(* Logix 5000 project; controller reports 1756-L63 rev 20.11; software revision 20.04; part 51 of 52 *)

        [192].log_data[2].total := 459.251, [192].log_data[2].time := 3600.0, [192].log_data[2].minminute := 7, [192].log_data[2].valid := 1, [192].log_data[3].time := 3600.0, [192].log_data[3].valid := 1, [192].log_data[4].time := 3600.0, [192].log_data[4].valid := 1, [192].log_data[5].max := 1.0, [192].log_data[5].total := 245.0, [192].log_data[5].time := 3600.0, [192].log_data[5].maxminute := 1, [192].log_data[5].valid := 1, [192].log_data[6].time := 3600.0, [192].log_data[6].valid := 1, [192].log_data[7].time := 3600.0, [192].log_data[7].valid := 1, [192].log_data[8].max := 1.0, [192].log_data[8].total := 3412.249, [192].log_data[8].time := 3600.0, [192].log_data[8].maxminute := 3, [192].log_data[8].valid := 1, [192].log_data[9].max := 1.0, [192].log_data[9].total := 3408.749, [192].log_data[9].time := 3600.0, [192].log_data[9].maxminute := 3, [192].log_data[9].valid := 1, [192].log_data[10].min := 1.0, [192].log_data[10].max := 1.0, [192].log_data[10].total := 3600.0, [192].log_data[10].time := 3600.0, [192].log_data[10].valid := 1, [192].log_data[11].time := 3600.0, [192].log_data[11].valid := 1, [192].log_data[12].min := 1.0, [192].log_data[12].max := 1.0, [192].log_data[12].total := 3600.0, [192].log_data[12].time := 3600.0, [192].log_data[12].valid := 1, [192].log_data[13].min := 1.0, [192].log_data[13].max := 1.0, [192].log_data[13].total := 3600.0, [192].log_data[13].time := 3600.0, [192].log_data[13].valid := 1, [192].log_data[14].time := 3600.0, [192].log_data[14].valid := 1, [192].log_data[15].time := 3600.0, [192].log_data[15].valid := 1, [192].log_data[16].time := 3600.0, [192].log_data[16].valid := 1, [192].log_data[17].min := 1.0, [192].log_data[17].max := 1.0, [192].log_data[17].total := 3600.0, [192].log_data[17].time := 3600.0, [192].log_data[17].valid := 1, [192].log_data[18].time := 3600.0, [192].log_data[18].valid := 1, [192].log_data[19].time := 3600.0, [192].log_data[19].valid := 1, [192].log_data[20].time := 3600.0,
        [192].log_data[20].valid := 1, [192].log_data[21].min := 1.0, [192].log_data[21].max := 1.0, [192].log_data[21].total := 3600.0, [192].log_data[21].time := 3600.0, [192].log_data[21].valid := 1, [192].log_data[22].time := 3600.0, [192].log_data[22].valid := 1, [192].log_data[23].time := 3600.0, [192].log_data[23].valid := 1, [192].log_data[24].time := 3600.0, [192].log_data[24].valid := 1, [192].log_data[25].time := 3600.0, [192].log_data[25].valid := 1, [192].log_data[26].time := 3600.0, [192].log_data[26].valid := 1, [192].log_data[27].time := 3600.0, [192].log_data[27].valid := 1, [192].log_data[28].time := 3600.0, [192].log_data[28].valid := 1, [192].log_data[29].min := 1.0, [192].log_data[29].max := 1.0, [192].log_data[29].total := 3600.0, [192].log_data[29].time := 3600.0, [192].log_data[29].valid := 1, [192].log_data[30].min := 1.0, [192].log_data[30].max := 1.0, [192].log_data[30].total := 3600.0, [192].log_data[30].time := 3600.0, [192].log_data[30].valid := 1, [192].log_data[31].max := 1.0, [192].log_data[31].total := 1629.998, [192].log_data[31].time := 3600.0, [192].log_data[31].maxminute := 5, [192].log_data[31].valid := 1, [192].log_data[32].max := 1.0, [192].log_data[32].total := 1245.496, [192].log_data[32].time := 3600.0, [192].log_data[32].maxminute := 3, [192].log_data[32].valid := 1, [192].log_data[33].time := 3600.0, [192].log_data[33].valid := 1, [192].log_data[34].time := 3600.0, [192].log_data[34].valid := 1, [192].log_data[35].max := 1.0, [192].log_data[35].total := 1309.247, [192].log_data[35].time := 3600.0, [192].log_data[35].maxminute := 3, [192].log_data[35].valid := 1, [192].log_data[36].max := 1.0, [192].log_data[36].total := 1629.7471, [192].log_data[36].time := 3600.0, [192].log_data[36].maxminute := 8, [192].log_data[36].valid := 1, [192].log_data[37].max := 7.618002, [192].log_data[37].total := 2978.067, [192].log_data[37].time := 3600.0, [192].log_data[37].minminute := 6, [192].log_data[37].maxminute := 1, [192].log_data[37].valid := 1,
        [192].log_data[38].time := 3600.0, [192].log_data[38].valid := 1, [192].log_data[39].min := 0.9956484, [192].log_data[39].max := 1.0215589, [192].log_data[39].total := 3607.7732, [192].log_data[39].time := 3600.0, [192].log_data[39].minminute := 25, [192].log_data[39].maxminute := 5, [192].log_data[39].valid := 1, [192].log_data[40].min := 7.5497513, [192].log_data[40].max := 7.5849276, [192].log_data[40].total := 27261.969, [192].log_data[40].time := 3600.0, [192].log_data[40].minminute := 39, [192].log_data[40].maxminute := 41, [192].log_data[40].valid := 1, [192].log_data[41].min := 0.071613036, [192].log_data[41].max := 0.10262695, [192].log_data[41].total := 306.5022, [192].log_data[41].time := 3600.0, [192].log_data[41].minminute := 38, [192].log_data[41].maxminute := 14, [192].log_data[41].valid := 1, [192].log_data[42].min := 2.2922316, [192].log_data[42].max := 2.2978847, [192].log_data[42].total := 8264.105, [192].log_data[42].time := 3600.0, [192].log_data[42].minminute := 46, [192].log_data[42].maxminute := 48, [192].log_data[42].valid := 1, [192].log_data[43].min := -0.26000214, [192].log_data[43].max := -0.23999786, [192].log_data[43].total := -935.0287, [192].log_data[43].time := 3600.0, [192].log_data[43].maxminute := 2, [192].log_data[43].valid := 1, [192].log_data[44].min := -0.30000305, [192].log_data[44].max := -0.27999878, [192].log_data[44].total := -1008.2222, [192].log_data[44].time := 3600.0, [192].log_data[44].valid := 1, [192].log_data[45].time := 3600.0, [192].log_data[45].valid := 1, [192].log_data[46].time := 3600.0, [192].log_data[46].valid := 1, [192].log_data[47].time := 3600.0, [192].log_data[47].valid := 1, [192].log_data[48].min := 6.583527, [192].log_data[48].max := 6.9622126, [192].log_data[48].total := 24239.32, [192].log_data[48].time := 3600.0, [192].log_data[48].minminute := 30, [192].log_data[48].maxminute := 7, [192].log_data[48].valid := 1, [192].log_data[49].min := 6.6613107, [192].log_data[49].max := 9.357373, [192].log_data[49].total := 28408.674, [192].log_data[49].time := 3600.0, [192].log_data[49].minminute := 28, [192].log_data[49].maxminute := 1,
        [192].log_data[49].valid := 1, [192].log_data[50].min := 2.0446687, [192].log_data[50].max := 2.150784, [192].log_data[50].total := 7503.921, [192].log_data[50].time := 3600.0, [192].log_data[50].minminute := 59, [192].log_data[50].maxminute := 3, [192].log_data[50].valid := 1, [192].log_data[51].time := 3600.0, [192].log_data[51].valid := 1, [192].log_data[52].min := -3.9399948, [192].log_data[52].max := 0.13999939, [192].log_data[52].total := -7269.7427, [192].log_data[52].time := 3600.0, [192].log_data[52].minminute := 3, [192].log_data[52].maxminute := 4, [192].log_data[52].valid := 1, [192].log_data[53].min := -3.659996, [192].log_data[53].max := 0.22000122, [192].log_data[53].total := -6986.5464, [192].log_data[53].time := 3600.0, [192].log_data[53].minminute := 3, [192].log_data[53].maxminute := 18, [192].log_data[53].valid := 1, [192].log_data[54].max := 0.52900004, [192].log_data[54].total := 1137.4148, [192].log_data[54].time := 3600.0, [192].log_data[54].maxminute := 26, [192].log_data[54].valid := 1, [192].log_data[55].max := 0.528, [192].log_data[55].total := 1164.4391, [192].log_data[55].time := 3600.0, [192].log_data[55].maxminute := 19, [192].log_data[55].valid := 1, [192].log_data[56].min := 0.16024561, [192].log_data[56].max := 0.16067745, [192].log_data[56].total := 577.62604, [192].log_data[56].time := 3600.0, [192].log_data[56].minminute := 30, [192].log_data[56].maxminute := 2, [192].log_data[56].valid := 1, [192].log_data[57].min := 0.33023393, [192].log_data[57].max := 0.33223614, [192].log_data[57].total := 1192.6987, [192].log_data[57].time := 3600.0, [192].log_data[57].minminute := 47, [192].log_data[57].maxminute := 2, [192].log_data[57].valid := 1, [192].log_data[58].time := 3600.0, [192].log_data[58].valid := 1, [192].log_data[59].time := 3600.0, [192].log_data[59].valid := 1, [192].log_data[60].valid := 1, [192].log_data[61].valid := 1, [192].log_data[62].valid := 1, [192].log_data[63].valid := 1, [192].log_data[64].valid := 1, [192].log_data[65].valid := 1, [192].log_data[66].valid := 1, [192].log_data[67].valid := 1,
        [192].log_data[68].valid := 1, [192].log_data[69].valid := 1, [192].log_data[70].valid := 1, [192].log_data[71].valid := 1, [192].log_data[72].valid := 1, [192].log_data[73].valid := 1, [192].log_data[74].valid := 1, [192].log_data[75].valid := 1, [192].log_data[76].valid := 1, [192].log_data[77].valid := 1, [192].log_data[78].valid := 1, [192].log_data[79].valid := 1, [192].log_data[80].valid := 1, [192].log_data[81].valid := 1, [192].log_data[82].valid := 1, [192].log_data[83].valid := 1, [192].log_data[84].valid := 1, [192].log_data[85].valid := 1, [192].log_data[86].valid := 1, [192].log_data[87].valid := 1, [192].log_data[88].valid := 1, [192].log_data[89].valid := 1, [192].log_data[90].valid := 1, [192].log_data[91].valid := 1, [192].log_data[92].valid := 1, [192].log_data[93].valid := 1, [192].log_data[94].valid := 1, [192].log_data[95].valid := 1, [192].log_data[96].valid := 1, [192].log_data[97].valid := 1, [192].log_data[98].valid := 1, [192].log_data[99].valid := 1, [192].log_data[100].valid := 1, [192].log_data[101].valid := 1, [192].log_data[102].valid := 1, [192].log_data[103].valid := 1, [192].log_data[104].valid := 1, [192].log_data[105].valid := 1, [192].log_data[106].valid := 1, [192].log_data[107].valid := 1, [192].log_data[108].valid := 1, [192].log_data[109].valid := 1, [192].log_data[110].valid := 1, [192].log_data[111].valid := 1, [192].log_data[112].valid := 1, [192].log_data[113].valid := 1, [192].log_data[114].valid := 1, [192].log_data[115].valid := 1, [192].log_data[116].valid := 1, [192].log_data[117].valid := 1, [192].log_data[118].valid := 1, [192].log_data[119].valid := 1, [192].log_data[120].valid := 1, [192].log_data[121].valid := 1, [192].log_data[122].valid := 1, [192].log_data[123].valid := 1, [192].log_data[124].valid := 1, [192].time.Year := 2023, [192].time.Month := 1, [192].time.Day := 12,
        [192].time.Hour := 19, [192].time.Minute := 59, [192].time.Second := 59, [193].log_data[0].min := 1.0, [193].log_data[0].max := 1.0, [193].log_data[0].total := 3600.0, [193].log_data[0].time := 3600.0, [193].log_data[0].valid := 1, [193].log_data[1].max := 1.0, [193].log_data[1].total := 593.5, [193].log_data[1].time := 3600.0, [193].log_data[1].maxminute := 21, [193].log_data[1].valid := 1, [193].log_data[2].max := 1.0, [193].log_data[2].total := 590.0, [193].log_data[2].time := 3600.0, [193].log_data[2].maxminute := 21, [193].log_data[2].valid := 1, [193].log_data[3].time := 3600.0, [193].log_data[3].valid := 1, [193].log_data[4].time := 3600.0, [193].log_data[4].valid := 1, [193].log_data[5].max := 1.0, [193].log_data[5].total := 233.5, [193].log_data[5].time := 3600.0, [193].log_data[5].maxminute := 24, [193].log_data[5].valid := 1, [193].log_data[6].time := 3600.0, [193].log_data[6].valid := 1, [193].log_data[7].time := 3600.0, [193].log_data[7].valid := 1, [193].log_data[8].min := 1.0, [193].log_data[8].max := 1.0, [193].log_data[8].total := 3600.0, [193].log_data[8].time := 3600.0, [193].log_data[8].valid := 1, [193].log_data[9].min := 1.0, [193].log_data[9].max := 1.0, [193].log_data[9].total := 3600.0, [193].log_data[9].time := 3600.0, [193].log_data[9].valid := 1, [193].log_data[10].min := 1.0, [193].log_data[10].max := 1.0, [193].log_data[10].total := 3600.0, [193].log_data[10].time := 3600.0, [193].log_data[10].valid := 1, [193].log_data[11].time := 3600.0, [193].log_data[11].valid := 1, [193].log_data[12].min := 1.0, [193].log_data[12].max := 1.0, [193].log_data[12].total := 3600.0, [193].log_data[12].time := 3600.0, [193].log_data[12].valid := 1, [193].log_data[13].min := 1.0, [193].log_data[13].max := 1.0, [193].log_data[13].total := 3600.0, [193].log_data[13].time := 3600.0, [193].log_data[13].valid := 1, [193].log_data[14].time := 3600.0, [193].log_data[14].valid := 1,
        [193].log_data[15].time := 3600.0, [193].log_data[15].valid := 1, [193].log_data[16].time := 3600.0, [193].log_data[16].valid := 1, [193].log_data[17].min := 1.0, [193].log_data[17].max := 1.0, [193].log_data[17].total := 3600.0, [193].log_data[17].time := 3600.0, [193].log_data[17].valid := 1, [193].log_data[18].time := 3600.0, [193].log_data[18].valid := 1, [193].log_data[19].time := 3600.0, [193].log_data[19].valid := 1, [193].log_data[20].time := 3600.0, [193].log_data[20].valid := 1, [193].log_data[21].min := 1.0, [193].log_data[21].max := 1.0, [193].log_data[21].total := 3600.0, [193].log_data[21].time := 3600.0, [193].log_data[21].valid := 1, [193].log_data[22].time := 3600.0, [193].log_data[22].valid := 1, [193].log_data[23].time := 3600.0, [193].log_data[23].valid := 1, [193].log_data[24].time := 3600.0, [193].log_data[24].valid := 1, [193].log_data[25].time := 3600.0, [193].log_data[25].valid := 1, [193].log_data[26].time := 3600.0, [193].log_data[26].valid := 1, [193].log_data[27].time := 3600.0, [193].log_data[27].valid := 1, [193].log_data[28].time := 3600.0, [193].log_data[28].valid := 1, [193].log_data[29].min := 1.0, [193].log_data[29].max := 1.0, [193].log_data[29].total := 3600.0, [193].log_data[29].time := 3600.0, [193].log_data[29].valid := 1, [193].log_data[30].min := 1.0, [193].log_data[30].max := 1.0, [193].log_data[30].total := 3600.0, [193].log_data[30].time := 3600.0, [193].log_data[30].valid := 1, [193].log_data[31].max := 1.0, [193].log_data[31].total := 1627.749, [193].log_data[31].time := 3600.0, [193].log_data[31].maxminute := 8, [193].log_data[31].valid := 1, [193].log_data[32].max := 1.0, [193].log_data[32].total := 1531.749, [193].log_data[32].time := 3600.0, [193].log_data[32].minminute := 7, [193].log_data[32].valid := 1, [193].log_data[33].time := 3600.0, [193].log_data[33].valid := 1, [193].log_data[34].time := 3600.0, [193].log_data[34].valid := 1, [193].log_data[35].max := 1.0, [193].log_data[35].total := 1629.7471,
        [193].log_data[35].time := 3600.0, [193].log_data[35].maxminute := 1, [193].log_data[35].valid := 1, [193].log_data[36].max := 1.0, [193].log_data[36].total := 1462.2471, [193].log_data[36].time := 3600.0, [193].log_data[36].maxminute := 11, [193].log_data[36].valid := 1, [193].log_data[37].max := 7.019314, [193].log_data[37].total := 3636.593, [193].log_data[37].time := 3600.0, [193].log_data[37].maxminute := 23, [193].log_data[37].valid := 1, [193].log_data[38].time := 3600.0, [193].log_data[38].valid := 1, [193].log_data[39].min := 0.9957663, [193].log_data[39].max := 1.0214411, [193].log_data[39].total := 3612.8372, [193].log_data[39].time := 3600.0, [193].log_data[39].minminute := 12, [193].log_data[39].maxminute := 24, [193].log_data[39].valid := 1, [193].log_data[40].min := 7.5588202, [193].log_data[40].max := 7.5835533, [193].log_data[40].total := 27258.096, [193].log_data[40].time := 3600.0, [193].log_data[40].minminute := 20, [193].log_data[40].maxminute := 24, [193].log_data[40].valid := 1, [193].log_data[41].min := 0.058461428, [193].log_data[41].max := 0.08123121, [193].log_data[41].total := 243.92332, [193].log_data[41].time := 3600.0, [193].log_data[41].minminute := 58, [193].log_data[41].valid := 1, [193].log_data[42].min := 2.2928205, [193].log_data[42].max := 2.2980025, [193].log_data[42].total := 8264.203, [193].log_data[42].time := 3600.0, [193].log_data[42].minminute := 33, [193].log_data[42].maxminute := 26, [193].log_data[42].valid := 1, [193].log_data[43].min := -0.26000214, [193].log_data[43].max := -0.23999786, [193].log_data[43].total := -934.74786, [193].log_data[43].time := 3600.0, [193].log_data[43].valid := 1, [193].log_data[44].min := -0.30000305, [193].log_data[44].max := -0.27999878, [193].log_data[44].total := -1008.36926, [193].log_data[44].time := 3600.0, [193].log_data[44].minminute := 9, [193].log_data[44].valid := 1, [193].log_data[45].time := 3600.0, [193].log_data[45].valid := 1, [193].log_data[46].time := 3600.0, [193].log_data[46].valid := 1, [193].log_data[47].time := 3600.0, [193].log_data[47].valid := 1, [193].log_data[48].min := 6.5824285,
        [193].log_data[48].max := 6.9251137, [193].log_data[48].total := 24218.438, [193].log_data[48].time := 3600.0, [193].log_data[48].minminute := 52, [193].log_data[48].maxminute := 31, [193].log_data[48].valid := 1, [193].log_data[49].min := 6.6723037, [193].log_data[49].max := 9.375628, [193].log_data[49].total := 29557.203, [193].log_data[49].time := 3600.0, [193].log_data[49].minminute := 50, [193].log_data[49].maxminute := 17, [193].log_data[49].valid := 1, [193].log_data[50].min := 2.0114563, [193].log_data[50].max := 2.1175714, [193].log_data[50].total := 7445.1196, [193].log_data[50].time := 3600.0, [193].log_data[50].minminute := 24, [193].log_data[50].maxminute := 32, [193].log_data[50].valid := 1, [193].log_data[51].time := 3600.0, [193].log_data[51].valid := 1, [193].log_data[52].min := -2.8199997, [193].log_data[52].max := 0.13999939, [193].log_data[52].total := -7697.88, [193].log_data[52].time := 3600.0, [193].log_data[52].minminute := 8, [193].log_data[52].maxminute := 7, [193].log_data[52].valid := 1, [193].log_data[53].min := -2.4800034, [193].log_data[53].max := 0.22000122, [193].log_data[53].total := -7055.2607, [193].log_data[53].time := 3600.0, [193].log_data[53].minminute := 3, [193].log_data[53].maxminute := 32, [193].log_data[53].valid := 1, [193].log_data[54].max := 0.536, [193].log_data[54].total := 1254.7595, [193].log_data[54].time := 3600.0, [193].log_data[54].minminute := 7, [193].log_data[54].maxminute := 8, [193].log_data[54].valid := 1, [193].log_data[55].max := 0.5365, [193].log_data[55].total := 1225.1177, [193].log_data[55].time := 3600.0, [193].log_data[55].maxminute := 22, [193].log_data[55].valid := 1, [193].log_data[56].min := 0.16024561, [193].log_data[56].max := 0.1607167, [193].log_data[56].total := 577.5824, [193].log_data[56].time := 3600.0, [193].log_data[56].minminute := 55, [193].log_data[56].valid := 1, [193].log_data[57].min := 0.32854584, [193].log_data[57].max := 0.33066577, [193].log_data[57].total := 1189.0582, [193].log_data[57].time := 3600.0, [193].log_data[57].minminute := 59, [193].log_data[57].maxminute := 6, [193].log_data[57].valid := 1,
        [193].log_data[58].time := 3600.0, [193].log_data[58].valid := 1, [193].log_data[59].time := 3600.0, [193].log_data[59].valid := 1, [193].log_data[60].valid := 1, [193].log_data[61].valid := 1, [193].log_data[62].valid := 1, [193].log_data[63].valid := 1, [193].log_data[64].valid := 1, [193].log_data[65].valid := 1, [193].log_data[66].valid := 1, [193].log_data[67].valid := 1, [193].log_data[68].valid := 1, [193].log_data[69].valid := 1, [193].log_data[70].valid := 1, [193].log_data[71].valid := 1, [193].log_data[72].valid := 1, [193].log_data[73].valid := 1, [193].log_data[74].valid := 1, [193].log_data[75].valid := 1, [193].log_data[76].valid := 1, [193].log_data[77].valid := 1, [193].log_data[78].valid := 1, [193].log_data[79].valid := 1, [193].log_data[80].valid := 1, [193].log_data[81].valid := 1, [193].log_data[82].valid := 1, [193].log_data[83].valid := 1, [193].log_data[84].valid := 1, [193].log_data[85].valid := 1, [193].log_data[86].valid := 1, [193].log_data[87].valid := 1, [193].log_data[88].valid := 1, [193].log_data[89].valid := 1, [193].log_data[90].valid := 1, [193].log_data[91].valid := 1, [193].log_data[92].valid := 1, [193].log_data[93].valid := 1, [193].log_data[94].valid := 1, [193].log_data[95].valid := 1, [193].log_data[96].valid := 1, [193].log_data[97].valid := 1, [193].log_data[98].valid := 1, [193].log_data[99].valid := 1, [193].log_data[100].valid := 1, [193].log_data[101].valid := 1, [193].log_data[102].valid := 1, [193].log_data[103].valid := 1, [193].log_data[104].valid := 1, [193].log_data[105].valid := 1, [193].log_data[106].valid := 1, [193].log_data[107].valid := 1, [193].log_data[108].valid := 1, [193].log_data[109].valid := 1, [193].log_data[110].valid := 1, [193].log_data[111].valid := 1, [193].log_data[112].valid := 1, [193].log_data[113].valid := 1, [193].log_data[114].valid := 1, [193].log_data[115].valid := 1,
        [193].log_data[116].valid := 1, [193].log_data[117].valid := 1, [193].log_data[118].valid := 1, [193].log_data[119].valid := 1, [193].log_data[120].valid := 1, [193].log_data[121].valid := 1, [193].log_data[122].valid := 1, [193].log_data[123].valid := 1, [193].log_data[124].valid := 1, [193].time.Year := 2023, [193].time.Month := 1, [193].time.Day := 12, [193].time.Hour := 20, [193].time.Minute := 59, [193].time.Second := 59, [194].log_data[0].min := 1.0, [194].log_data[0].max := 1.0, [194].log_data[0].total := 3600.0, [194].log_data[0].time := 3600.0, [194].log_data[0].valid := 1, [194].log_data[1].max := 1.0, [194].log_data[1].total := 582.5, [194].log_data[1].time := 3600.0, [194].log_data[1].maxminute := 30, [194].log_data[1].valid := 1, [194].log_data[2].max := 1.0, [194].log_data[2].total := 579.0, [194].log_data[2].time := 3600.0, [194].log_data[2].maxminute := 30, [194].log_data[2].valid := 1, [194].log_data[3].time := 3600.0, [194].log_data[3].valid := 1, [194].log_data[4].time := 3600.0, [194].log_data[4].valid := 1, [194].log_data[5].max := 1.0, [194].log_data[5].total := 246.0, [194].log_data[5].time := 3600.0, [194].log_data[5].maxminute := 32, [194].log_data[5].valid := 1, [194].log_data[6].time := 3600.0, [194].log_data[6].valid := 1, [194].log_data[7].time := 3600.0, [194].log_data[7].valid := 1, [194].log_data[8].min := 1.0, [194].log_data[8].max := 1.0, [194].log_data[8].total := 3600.0, [194].log_data[8].time := 3600.0, [194].log_data[8].valid := 1, [194].log_data[9].min := 1.0, [194].log_data[9].max := 1.0, [194].log_data[9].total := 3600.0, [194].log_data[9].time := 3600.0, [194].log_data[9].valid := 1, [194].log_data[10].min := 1.0, [194].log_data[10].max := 1.0, [194].log_data[10].total := 3600.0, [194].log_data[10].time := 3600.0, [194].log_data[10].valid := 1, [194].log_data[11].time := 3600.0, [194].log_data[11].valid := 1,
        [194].log_data[12].min := 1.0, [194].log_data[12].max := 1.0, [194].log_data[12].total := 3600.0, [194].log_data[12].time := 3600.0, [194].log_data[12].valid := 1, [194].log_data[13].min := 1.0, [194].log_data[13].max := 1.0, [194].log_data[13].total := 3600.0, [194].log_data[13].time := 3600.0, [194].log_data[13].valid := 1, [194].log_data[14].time := 3600.0, [194].log_data[14].valid := 1, [194].log_data[15].time := 3600.0, [194].log_data[15].valid := 1, [194].log_data[16].time := 3600.0, [194].log_data[16].valid := 1, [194].log_data[17].min := 1.0, [194].log_data[17].max := 1.0, [194].log_data[17].total := 3600.0, [194].log_data[17].time := 3600.0, [194].log_data[17].valid := 1, [194].log_data[18].time := 3600.0, [194].log_data[18].valid := 1, [194].log_data[19].time := 3600.0, [194].log_data[19].valid := 1, [194].log_data[20].time := 3600.0, [194].log_data[20].valid := 1, [194].log_data[21].min := 1.0, [194].log_data[21].max := 1.0, [194].log_data[21].total := 3600.0, [194].log_data[21].time := 3600.0, [194].log_data[21].valid := 1, [194].log_data[22].time := 3600.0, [194].log_data[22].valid := 1, [194].log_data[23].time := 3600.0, [194].log_data[23].valid := 1, [194].log_data[24].time := 3600.0, [194].log_data[24].valid := 1, [194].log_data[25].time := 3600.0, [194].log_data[25].valid := 1, [194].log_data[26].time := 3600.0, [194].log_data[26].valid := 1, [194].log_data[27].time := 3600.0, [194].log_data[27].valid := 1, [194].log_data[28].time := 3600.0, [194].log_data[28].valid := 1, [194].log_data[29].min := 1.0, [194].log_data[29].max := 1.0, [194].log_data[29].total := 3600.0, [194].log_data[29].time := 3600.0, [194].log_data[29].valid := 1, [194].log_data[30].min := 1.0, [194].log_data[30].max := 1.0, [194].log_data[30].total := 3600.0, [194].log_data[30].time := 3600.0, [194].log_data[30].valid := 1, [194].log_data[31].max := 1.0, [194].log_data[31].total := 1440.7471, [194].log_data[31].time := 3600.0, [194].log_data[31].valid := 1,
        [194].log_data[32].max := 1.0, [194].log_data[32].total := 1629.7471, [194].log_data[32].time := 3600.0, [194].log_data[32].maxminute := 1, [194].log_data[32].valid := 1, [194].log_data[33].time := 3600.0, [194].log_data[33].valid := 1, [194].log_data[34].time := 3600.0, [194].log_data[34].valid := 1, [194].log_data[35].max := 1.0, [194].log_data[35].total := 1629.998, [194].log_data[35].time := 3600.0, [194].log_data[35].maxminute := 4, [194].log_data[35].valid := 1, [194].log_data[36].max := 1.0, [194].log_data[36].total := 1440.2471, [194].log_data[36].time := 3600.0, [194].log_data[36].minminute := 2, [194].log_data[36].valid := 1, [194].log_data[37].max := 7.519464, [194].log_data[37].total := 3829.7646, [194].log_data[37].time := 3600.0, [194].log_data[37].maxminute := 31, [194].log_data[37].valid := 1, [194].log_data[38].time := 3600.0, [194].log_data[38].valid := 1, [194].log_data[39].min := 0.9983573, [194].log_data[39].max := 1.0212055, [194].log_data[39].total := 3620.0103, [194].log_data[39].time := 3600.0, [194].log_data[39].minminute := 16, [194].log_data[39].maxminute := 36, [194].log_data[39].valid := 1, [194].log_data[40].min := 7.563218, [194].log_data[40].max := 7.5791564, [194].log_data[40].total := 27266.686, [194].log_data[40].time := 3600.0, [194].log_data[40].minminute := 7, [194].log_data[40].maxminute := 20, [194].log_data[40].valid := 1, [194].log_data[41].min := 0.052376464, [194].log_data[41].max := 0.08123121, [194].log_data[41].total := 235.2598, [194].log_data[41].time := 3600.0, [194].log_data[41].minminute := 7, [194].log_data[41].maxminute := 34, [194].log_data[41].valid := 1, [194].log_data[42].min := 2.2928205, [194].log_data[42].max := 2.2978847, [194].log_data[42].total := 8264.382, [194].log_data[42].time := 3600.0, [194].log_data[42].minminute := 20, [194].log_data[42].maxminute := 26, [194].log_data[42].valid := 1, [194].log_data[43].min := -0.26000214, [194].log_data[43].max := -0.23999786, [194].log_data[43].total := -931.67035, [194].log_data[43].time := 3600.0, [194].log_data[43].valid := 1, [194].log_data[44].min := -0.30000305,
        [194].log_data[44].max := -0.27999878, [194].log_data[44].total := -1007.9264, [194].log_data[44].time := 3600.0, [194].log_data[44].minminute := 9, [194].log_data[44].valid := 1, [194].log_data[45].time := 3600.0, [194].log_data[45].valid := 1, [194].log_data[46].time := 3600.0, [194].log_data[46].valid := 1, [194].log_data[47].time := 3600.0, [194].log_data[47].valid := 1, [194].log_data[48].min := 6.599191, [194].log_data[48].max := 6.9251137, [194].log_data[48].total := 24330.205, [194].log_data[48].time := 3600.0, [194].log_data[48].minminute := 59, [194].log_data[48].maxminute := 35, [194].log_data[48].valid := 1, [194].log_data[49].min := 6.62853, [194].log_data[49].max := 9.253535, [194].log_data[49].total := 29404.414, [194].log_data[49].time := 3600.0, [194].log_data[49].minminute := 58, [194].log_data[49].maxminute := 32, [194].log_data[49].valid := 1, [194].log_data[50].min := 2.0350113, [194].log_data[50].max := 2.1478395, [194].log_data[50].total := 7529.1016, [194].log_data[50].time := 3600.0, [194].log_data[50].minminute := 31, [194].log_data[50].maxminute := 39, [194].log_data[50].valid := 1, [194].log_data[51].time := 3600.0, [194].log_data[51].valid := 1, [194].log_data[52].min := -2.8199997, [194].log_data[52].max := 0.13999939, [194].log_data[52].total := -7484.4546, [194].log_data[52].time := 3600.0, [194].log_data[52].minminute := 33, [194].log_data[52].valid := 1, [194].log_data[53].min := -2.4800034, [194].log_data[53].max := 0.22000122, [194].log_data[53].total := -7043.564, [194].log_data[53].time := 3600.0, [194].log_data[53].minminute := 4, [194].log_data[53].maxminute := 45, [194].log_data[53].valid := 1, [194].log_data[54].max := 0.532, [194].log_data[54].total := 1217.1526, [194].log_data[54].time := 3600.0, [194].log_data[54].maxminute := 43, [194].log_data[54].valid := 1, [194].log_data[55].max := 0.56049997, [194].log_data[55].total := 1217.6139, [194].log_data[55].time := 3600.0, [194].log_data[55].minminute := 2, [194].log_data[55].maxminute := 56, [194].log_data[55].valid := 1, [194].log_data[56].min := 0.16032413, [194].log_data[56].max := 0.16067745,
        [194].log_data[56].total := 577.6923, [194].log_data[56].time := 3600.0, [194].log_data[56].maxminute := 3, [194].log_data[56].valid := 1, [194].log_data[57].min := 0.32823178, [194].log_data[57].max := 0.3287814, [194].log_data[57].total := 1182.377, [194].log_data[57].time := 3600.0, [194].log_data[57].minminute := 44, [194].log_data[57].valid := 1, [194].log_data[58].time := 3600.0, [194].log_data[58].valid := 1, [194].log_data[59].time := 3600.0, [194].log_data[59].valid := 1, [194].log_data[60].valid := 1, [194].log_data[61].valid := 1, [194].log_data[62].valid := 1, [194].log_data[63].valid := 1, [194].log_data[64].valid := 1, [194].log_data[65].valid := 1, [194].log_data[66].valid := 1, [194].log_data[67].valid := 1, [194].log_data[68].valid := 1, [194].log_data[69].valid := 1, [194].log_data[70].valid := 1, [194].log_data[71].valid := 1, [194].log_data[72].valid := 1, [194].log_data[73].valid := 1, [194].log_data[74].valid := 1, [194].log_data[75].valid := 1, [194].log_data[76].valid := 1, [194].log_data[77].valid := 1, [194].log_data[78].valid := 1, [194].log_data[79].valid := 1, [194].log_data[80].valid := 1, [194].log_data[81].valid := 1, [194].log_data[82].valid := 1, [194].log_data[83].valid := 1, [194].log_data[84].valid := 1, [194].log_data[85].valid := 1, [194].log_data[86].valid := 1, [194].log_data[87].valid := 1, [194].log_data[88].valid := 1, [194].log_data[89].valid := 1, [194].log_data[90].valid := 1, [194].log_data[91].valid := 1, [194].log_data[92].valid := 1, [194].log_data[93].valid := 1, [194].log_data[94].valid := 1, [194].log_data[95].valid := 1, [194].log_data[96].valid := 1, [194].log_data[97].valid := 1, [194].log_data[98].valid := 1, [194].log_data[99].valid := 1, [194].log_data[100].valid := 1, [194].log_data[101].valid := 1, [194].log_data[102].valid := 1, [194].log_data[103].valid := 1, [194].log_data[104].valid := 1, [194].log_data[105].valid := 1,
        [194].log_data[106].valid := 1, [194].log_data[107].valid := 1, [194].log_data[108].valid := 1, [194].log_data[109].valid := 1, [194].log_data[110].valid := 1, [194].log_data[111].valid := 1, [194].log_data[112].valid := 1, [194].log_data[113].valid := 1, [194].log_data[114].valid := 1, [194].log_data[115].valid := 1, [194].log_data[116].valid := 1, [194].log_data[117].valid := 1, [194].log_data[118].valid := 1, [194].log_data[119].valid := 1, [194].log_data[120].valid := 1, [194].log_data[121].valid := 1, [194].log_data[122].valid := 1, [194].log_data[123].valid := 1, [194].log_data[124].valid := 1, [194].time.Year := 2023, [194].time.Month := 1, [194].time.Day := 12, [194].time.Hour := 21, [194].time.Minute := 59, [194].time.Second := 59, [195].log_data[0].min := 1.0, [195].log_data[0].max := 1.0, [195].log_data[0].total := 3600.0, [195].log_data[0].time := 3600.0, [195].log_data[0].valid := 1, [195].log_data[1].max := 1.0, [195].log_data[1].total := 595.5, [195].log_data[1].time := 3600.0, [195].log_data[1].maxminute := 34, [195].log_data[1].valid := 1, [195].log_data[2].max := 1.0, [195].log_data[2].total := 592.0, [195].log_data[2].time := 3600.0, [195].log_data[2].maxminute := 34, [195].log_data[2].valid := 1, [195].log_data[3].time := 3600.0, [195].log_data[3].valid := 1, [195].log_data[4].time := 3600.0, [195].log_data[4].valid := 1, [195].log_data[5].max := 1.0, [195].log_data[5].total := 239.5, [195].log_data[5].time := 3600.0, [195].log_data[5].maxminute := 36, [195].log_data[5].valid := 1, [195].log_data[6].time := 3600.0, [195].log_data[6].valid := 1, [195].log_data[7].time := 3600.0, [195].log_data[7].valid := 1, [195].log_data[8].min := 1.0, [195].log_data[8].max := 1.0, [195].log_data[8].total := 3600.0, [195].log_data[8].time := 3600.0, [195].log_data[8].valid := 1, [195].log_data[9].min := 1.0, [195].log_data[9].max := 1.0,
        [195].log_data[9].total := 3600.0, [195].log_data[9].time := 3600.0, [195].log_data[9].valid := 1, [195].log_data[10].min := 1.0, [195].log_data[10].max := 1.0, [195].log_data[10].total := 3600.0, [195].log_data[10].time := 3600.0, [195].log_data[10].valid := 1, [195].log_data[11].time := 3600.0, [195].log_data[11].valid := 1, [195].log_data[12].min := 1.0, [195].log_data[12].max := 1.0, [195].log_data[12].total := 3600.0, [195].log_data[12].time := 3600.0, [195].log_data[12].valid := 1, [195].log_data[13].min := 1.0, [195].log_data[13].max := 1.0, [195].log_data[13].total := 3600.0, [195].log_data[13].time := 3600.0, [195].log_data[13].valid := 1, [195].log_data[14].time := 3600.0, [195].log_data[14].valid := 1, [195].log_data[15].time := 3600.0, [195].log_data[15].valid := 1, [195].log_data[16].time := 3600.0, [195].log_data[16].valid := 1, [195].log_data[17].min := 1.0, [195].log_data[17].max := 1.0, [195].log_data[17].total := 3600.0, [195].log_data[17].time := 3600.0, [195].log_data[17].valid := 1, [195].log_data[18].time := 3600.0, [195].log_data[18].valid := 1, [195].log_data[19].time := 3600.0, [195].log_data[19].valid := 1, [195].log_data[20].time := 3600.0, [195].log_data[20].valid := 1, [195].log_data[21].min := 1.0, [195].log_data[21].max := 1.0, [195].log_data[21].total := 3600.0, [195].log_data[21].time := 3600.0, [195].log_data[21].valid := 1, [195].log_data[22].time := 3600.0, [195].log_data[22].valid := 1, [195].log_data[23].time := 3600.0, [195].log_data[23].valid := 1, [195].log_data[24].time := 3600.0, [195].log_data[24].valid := 1, [195].log_data[25].time := 3600.0, [195].log_data[25].valid := 1, [195].log_data[26].time := 3600.0, [195].log_data[26].valid := 1, [195].log_data[27].time := 3600.0, [195].log_data[27].valid := 1, [195].log_data[28].time := 3600.0, [195].log_data[28].valid := 1, [195].log_data[29].min := 1.0, [195].log_data[29].max := 1.0, [195].log_data[29].total := 3600.0, [195].log_data[29].time := 3600.0,
        [195].log_data[29].valid := 1, [195].log_data[30].min := 1.0, [195].log_data[30].max := 1.0, [195].log_data[30].total := 3600.0, [195].log_data[30].time := 3600.0, [195].log_data[30].valid := 1, [195].log_data[31].max := 1.0, [195].log_data[31].total := 1440.998, [195].log_data[31].time := 3600.0, [195].log_data[31].minminute := 3, [195].log_data[31].valid := 1, [195].log_data[32].max := 1.0, [195].log_data[32].total := 1630.249, [195].log_data[32].time := 3600.0, [195].log_data[32].maxminute := 4, [195].log_data[32].valid := 1, [195].log_data[33].time := 3600.0, [195].log_data[33].valid := 1, [195].log_data[34].time := 3600.0, [195].log_data[34].valid := 1, [195].log_data[35].max := 1.0, [195].log_data[35].total := 1629.7471, [195].log_data[35].time := 3600.0, [195].log_data[35].maxminute := 7, [195].log_data[35].valid := 1, [195].log_data[36].max := 1.0, [195].log_data[36].total := 1443.749, [195].log_data[36].time := 3600.0, [195].log_data[36].minminute := 5, [195].log_data[36].valid := 1, [195].log_data[37].max := 7.008321, [195].log_data[37].total := 3647.1792, [195].log_data[37].time := 3600.0, [195].log_data[37].maxminute := 35, [195].log_data[37].valid := 1, [195].log_data[38].time := 3600.0, [195].log_data[38].valid := 1, [195].log_data[39].min := 0.997415, [195].log_data[39].max := 1.0223833, [195].log_data[39].total := 3626.4546, [195].log_data[39].time := 3600.0, [195].log_data[39].minminute := 38, [195].log_data[39].maxminute := 40, [195].log_data[39].valid := 1, [195].log_data[40].min := 7.5643167, [195].log_data[40].max := 7.5777817, [195].log_data[40].total := 27267.686, [195].log_data[40].time := 3600.0, [195].log_data[40].minminute := 2, [195].log_data[40].valid := 1, [195].log_data[41].min := 0.05747998, [195].log_data[41].max := 0.08633472, [195].log_data[41].total := 263.88226, [195].log_data[41].time := 3600.0, [195].log_data[41].minminute := 8, [195].log_data[41].maxminute := 43, [195].log_data[41].valid := 1, [195].log_data[42].min := 2.2923493, [195].log_data[42].max := 2.2980025, [195].log_data[42].total := 8264.417,
        [195].log_data[42].time := 3600.0, [195].log_data[42].minminute := 28, [195].log_data[42].maxminute := 5, [195].log_data[42].valid := 1, [195].log_data[43].min := -0.26000214, [195].log_data[43].max := -0.23999786, [195].log_data[43].total := -935.618, [195].log_data[43].time := 3600.0, [195].log_data[43].valid := 1, [195].log_data[44].min := -0.30000305, [195].log_data[44].max := -0.27999878, [195].log_data[44].total := -1010.45667, [195].log_data[44].time := 3600.0, [195].log_data[44].minminute := 3, [195].log_data[44].valid := 1, [195].log_data[45].time := 3600.0, [195].log_data[45].valid := 1, [195].log_data[46].time := 3600.0, [195].log_data[46].valid := 1, [195].log_data[47].time := 3600.0, [195].log_data[47].valid := 1, [195].log_data[48].min := 6.5862756, [195].log_data[48].max := 6.940778, [195].log_data[48].total := 24259.021, [195].log_data[48].time := 3600.0, [195].log_data[48].minminute := 2, [195].log_data[48].maxminute := 42, [195].log_data[48].valid := 1, [195].log_data[49].min := 6.6885953, [195].log_data[49].max := 9.198378, [195].log_data[49].total := 28791.09, [195].log_data[49].time := 3600.0, [195].log_data[49].maxminute := 36, [195].log_data[49].valid := 1, [195].log_data[50].min := 2.0709326, [195].log_data[50].max := 2.1804633, [195].log_data[50].total := 7643.46, [195].log_data[50].time := 3600.0, [195].log_data[50].minminute := 35, [195].log_data[50].maxminute := 43, [195].log_data[50].valid := 1, [195].log_data[51].time := 3600.0, [195].log_data[51].valid := 1, [195].log_data[52].min := -2.9800034, [195].log_data[52].max := 0.13999939, [195].log_data[52].total := -7496.2583, [195].log_data[52].time := 3600.0, [195].log_data[52].minminute := 4, [195].log_data[52].maxminute := 14, [195].log_data[52].valid := 1, [195].log_data[53].min := -2.7200012, [195].log_data[53].max := 0.19999695, [195].log_data[53].total := -7053.963, [195].log_data[53].time := 3600.0, [195].log_data[53].minminute := 28, [195].log_data[53].maxminute := 6, [195].log_data[53].valid := 1, [195].log_data[54].max := 0.5335, [195].log_data[54].total := 1217.511, [195].log_data[54].time := 3600.0,
        [195].log_data[54].minminute := 3, [195].log_data[54].maxminute := 36, [195].log_data[54].valid := 1, [195].log_data[55].max := 0.575, [195].log_data[55].total := 1221.0226, [195].log_data[55].time := 3600.0, [195].log_data[55].minminute := 5, [195].log_data[55].maxminute := 28, [195].log_data[55].valid := 1, [195].log_data[56].min := 0.16024561, [195].log_data[56].max := 0.16075596, [195].log_data[56].total := 577.672, [195].log_data[56].time := 3600.0, [195].log_data[56].minminute := 29, [195].log_data[56].maxminute := 34, [195].log_data[56].valid := 1, [195].log_data[57].min := 0.3265829, [195].log_data[57].max := 0.32854584, [195].log_data[57].total := 1176.8693, [195].log_data[57].time := 3600.0, [195].log_data[57].minminute := 53, [195].log_data[57].valid := 1, [195].log_data[58].time := 3600.0, [195].log_data[58].valid := 1, [195].log_data[59].time := 3600.0, [195].log_data[59].valid := 1, [195].log_data[60].valid := 1, [195].log_data[61].valid := 1, [195].log_data[62].valid := 1, [195].log_data[63].valid := 1, [195].log_data[64].valid := 1, [195].log_data[65].valid := 1, [195].log_data[66].valid := 1, [195].log_data[67].valid := 1, [195].log_data[68].valid := 1, [195].log_data[69].valid := 1, [195].log_data[70].valid := 1, [195].log_data[71].valid := 1, [195].log_data[72].valid := 1, [195].log_data[73].valid := 1, [195].log_data[74].valid := 1, [195].log_data[75].valid := 1, [195].log_data[76].valid := 1, [195].log_data[77].valid := 1, [195].log_data[78].valid := 1, [195].log_data[79].valid := 1, [195].log_data[80].valid := 1, [195].log_data[81].valid := 1, [195].log_data[82].valid := 1, [195].log_data[83].valid := 1, [195].log_data[84].valid := 1, [195].log_data[85].valid := 1, [195].log_data[86].valid := 1, [195].log_data[87].valid := 1, [195].log_data[88].valid := 1, [195].log_data[89].valid := 1, [195].log_data[90].valid := 1, [195].log_data[91].valid := 1, [195].log_data[92].valid := 1, [195].log_data[93].valid := 1,
        [195].log_data[94].valid := 1, [195].log_data[95].valid := 1, [195].log_data[96].valid := 1, [195].log_data[97].valid := 1, [195].log_data[98].valid := 1, [195].log_data[99].valid := 1, [195].log_data[100].valid := 1, [195].log_data[101].valid := 1, [195].log_data[102].valid := 1, [195].log_data[103].valid := 1, [195].log_data[104].valid := 1, [195].log_data[105].valid := 1, [195].log_data[106].valid := 1, [195].log_data[107].valid := 1, [195].log_data[108].valid := 1, [195].log_data[109].valid := 1, [195].log_data[110].valid := 1, [195].log_data[111].valid := 1, [195].log_data[112].valid := 1, [195].log_data[113].valid := 1, [195].log_data[114].valid := 1, [195].log_data[115].valid := 1, [195].log_data[116].valid := 1, [195].log_data[117].valid := 1, [195].log_data[118].valid := 1, [195].log_data[119].valid := 1, [195].log_data[120].valid := 1, [195].log_data[121].valid := 1, [195].log_data[122].valid := 1, [195].log_data[123].valid := 1, [195].log_data[124].valid := 1, [195].time.Year := 2023, [195].time.Month := 1, [195].time.Day := 12, [195].time.Hour := 22, [195].time.Minute := 59, [195].time.Second := 59, [196].log_data[0].min := 1.0, [196].log_data[0].max := 1.0, [196].log_data[0].total := 3600.0, [196].log_data[0].time := 3600.0, [196].log_data[0].valid := 1, [196].log_data[1].max := 1.0, [196].log_data[1].total := 147.249, [196].log_data[1].time := 3600.0, [196].log_data[1].maxminute := 57, [196].log_data[1].valid := 1, [196].log_data[2].max := 1.0, [196].log_data[2].total := 143.749, [196].log_data[2].time := 3600.0, [196].log_data[2].maxminute := 57, [196].log_data[2].valid := 1, [196].log_data[3].time := 3600.0, [196].log_data[3].valid := 1, [196].log_data[4].time := 3600.0, [196].log_data[4].valid := 1, [196].log_data[5].max := 1.0, [196].log_data[5].total := 50.249, [196].log_data[5].time := 3600.0, [196].log_data[5].maxminute := 59,
        [196].log_data[5].valid := 1, [196].log_data[6].time := 3600.0, [196].log_data[6].valid := 1, [196].log_data[7].time := 3600.0, [196].log_data[7].valid := 1, [196].log_data[8].min := 1.0, [196].log_data[8].max := 1.0, [196].log_data[8].total := 3600.0, [196].log_data[8].time := 3600.0, [196].log_data[8].valid := 1, [196].log_data[9].min := 1.0, [196].log_data[9].max := 1.0, [196].log_data[9].total := 3600.0, [196].log_data[9].time := 3600.0, [196].log_data[9].valid := 1, [196].log_data[10].min := 1.0, [196].log_data[10].max := 1.0, [196].log_data[10].total := 3600.0, [196].log_data[10].time := 3600.0, [196].log_data[10].valid := 1, [196].log_data[11].time := 3600.0, [196].log_data[11].valid := 1, [196].log_data[12].min := 1.0, [196].log_data[12].max := 1.0, [196].log_data[12].total := 3600.0, [196].log_data[12].time := 3600.0, [196].log_data[12].valid := 1, [196].log_data[13].min := 1.0, [196].log_data[13].max := 1.0, [196].log_data[13].total := 3600.0, [196].log_data[13].time := 3600.0, [196].log_data[13].valid := 1, [196].log_data[14].time := 3600.0, [196].log_data[14].valid := 1, [196].log_data[15].time := 3600.0, [196].log_data[15].valid := 1, [196].log_data[16].time := 3600.0, [196].log_data[16].valid := 1, [196].log_data[17].min := 1.0, [196].log_data[17].max := 1.0, [196].log_data[17].total := 3600.0, [196].log_data[17].time := 3600.0, [196].log_data[17].valid := 1, [196].log_data[18].time := 3600.0, [196].log_data[18].valid := 1, [196].log_data[19].time := 3600.0, [196].log_data[19].valid := 1, [196].log_data[20].time := 3600.0, [196].log_data[20].valid := 1, [196].log_data[21].min := 1.0, [196].log_data[21].max := 1.0, [196].log_data[21].total := 3600.0, [196].log_data[21].time := 3600.0, [196].log_data[21].valid := 1, [196].log_data[22].time := 3600.0, [196].log_data[22].valid := 1, [196].log_data[23].time := 3600.0, [196].log_data[23].valid := 1, [196].log_data[24].time := 3600.0, [196].log_data[24].valid := 1,
        [196].log_data[25].time := 3600.0, [196].log_data[25].valid := 1, [196].log_data[26].time := 3600.0, [196].log_data[26].valid := 1, [196].log_data[27].time := 3600.0, [196].log_data[27].valid := 1, [196].log_data[28].time := 3600.0, [196].log_data[28].valid := 1, [196].log_data[29].min := 1.0, [196].log_data[29].max := 1.0, [196].log_data[29].total := 3600.0, [196].log_data[29].time := 3600.0, [196].log_data[29].valid := 1, [196].log_data[30].min := 1.0, [196].log_data[30].max := 1.0, [196].log_data[30].total := 3600.0, [196].log_data[30].time := 3600.0, [196].log_data[30].valid := 1, [196].log_data[31].max := 1.0, [196].log_data[31].total := 1466.998, [196].log_data[31].time := 3600.0, [196].log_data[31].minminute := 6, [196].log_data[31].valid := 1, [196].log_data[32].max := 1.0, [196].log_data[32].total := 1629.7471, [196].log_data[32].time := 3600.0, [196].log_data[32].maxminute := 7, [196].log_data[32].valid := 1, [196].log_data[33].time := 3600.0, [196].log_data[33].valid := 1, [196].log_data[34].time := 3600.0, [196].log_data[34].valid := 1, [196].log_data[35].max := 1.0, [196].log_data[35].total := 1526.2471, [196].log_data[35].time := 3600.0, [196].log_data[35].maxminute := 10, [196].log_data[35].valid := 1, [196].log_data[36].max := 1.0, [196].log_data[36].total := 1629.7471, [196].log_data[36].time := 3600.0, [196].log_data[36].valid := 1, [196].log_data[37].max := 7.646661, [196].log_data[37].total := 1097.6161, [196].log_data[37].time := 3600.0, [196].log_data[37].maxminute := 59, [196].log_data[37].valid := 1, [196].log_data[38].time := 3600.0, [196].log_data[38].valid := 1, [196].log_data[39].min := 1.0028327, [196].log_data[39].max := 1.0204989, [196].log_data[39].total := 3628.7998, [196].log_data[39].time := 3600.0, [196].log_data[39].minminute := 1, [196].log_data[39].maxminute := 59, [196].log_data[39].valid := 1, [196].log_data[40].min := 7.5527744, [196].log_data[40].max := 7.587675, [196].log_data[40].total := 27262.863, [196].log_data[40].time := 3600.0, [196].log_data[40].minminute := 2,
        [196].log_data[40].maxminute := 13, [196].log_data[40].valid := 1, [196].log_data[41].min := 0.045309816, [196].log_data[41].max := 0.072005615, [196].log_data[41].total := 215.19913, [196].log_data[41].time := 3600.0, [196].log_data[41].minminute := 38, [196].log_data[41].maxminute := 18, [196].log_data[41].valid := 1, [196].log_data[42].min := 2.2927027, [196].log_data[42].max := 2.2984736, [196].log_data[42].total := 8264.532, [196].log_data[42].time := 3600.0, [196].log_data[42].minminute := 28, [196].log_data[42].maxminute := 49, [196].log_data[42].valid := 1, [196].log_data[43].min := -0.26000214, [196].log_data[43].max := -0.23999786, [196].log_data[43].total := -935.9431, [196].log_data[43].time := 3600.0, [196].log_data[43].maxminute := 10, [196].log_data[43].valid := 1, [196].log_data[44].min := -0.30000305, [196].log_data[44].max := -0.27999878, [196].log_data[44].total := -1016.3021, [196].log_data[44].time := 3600.0, [196].log_data[44].valid := 1, [196].log_data[45].time := 3600.0, [196].log_data[45].valid := 1, [196].log_data[46].time := 3600.0, [196].log_data[46].valid := 1, [196].log_data[47].time := 3600.0, [196].log_data[47].valid := 1, [196].log_data[48].min := 6.586825, [196].log_data[48].max := 6.8162894, [196].log_data[48].total := 24217.527, [196].log_data[48].time := 3600.0, [196].log_data[48].minminute := 5, [196].log_data[48].maxminute := 59, [196].log_data[48].valid := 1, [196].log_data[49].min := 6.687418, [196].log_data[49].max := 9.361299, [196].log_data[49].total := 30686.113, [196].log_data[49].time := 3600.0, [196].log_data[49].minminute := 1, [196].log_data[49].maxminute := 57, [196].log_data[49].valid := 1, [196].log_data[50].min := 2.0794125, [196].log_data[50].max := 2.165506, [196].log_data[50].total := 7641.2354, [196].log_data[50].time := 3600.0, [196].log_data[50].minminute := 58, [196].log_data[50].valid := 1, [196].log_data[51].time := 3600.0, [196].log_data[51].valid := 1, [196].log_data[52].min := -2.9800034, [196].log_data[52].max := 0.11999512, [196].log_data[52].total := -7627.5664, [196].log_data[52].time := 3600.0, [196].log_data[52].minminute := 49,
        [196].log_data[52].maxminute := 6, [196].log_data[52].valid := 1, [196].log_data[53].min := -2.4800034, [196].log_data[53].max := 0.19999695, [196].log_data[53].total := -7256.613, [196].log_data[53].time := 3600.0, [196].log_data[53].minminute := 11, [196].log_data[53].maxminute := 9, [196].log_data[53].valid := 1, [196].log_data[54].max := 0.532, [196].log_data[54].total := 1229.739, [196].log_data[54].time := 3600.0, [196].log_data[54].minminute := 6, [196].log_data[54].maxminute := 50, [196].log_data[54].valid := 1, [196].log_data[55].max := 0.52, [196].log_data[55].total := 1250.6741, [196].log_data[55].time := 3600.0, [196].log_data[55].maxminute := 31, [196].log_data[55].valid := 1, [196].log_data[56].min := 0.16020635, [196].log_data[56].max := 0.1607167, [196].log_data[56].total := 577.64624, [196].log_data[56].time := 3600.0, [196].log_data[56].minminute := 5, [196].log_data[56].maxminute := 18, [196].log_data[56].valid := 1, [196].log_data[57].min := 0.32509112, [196].log_data[57].max := 0.32693627, [196].log_data[57].total := 1171.6685, [196].log_data[57].time := 3600.0, [196].log_data[57].minminute := 23, [196].log_data[57].valid := 1, [196].log_data[58].time := 3600.0, [196].log_data[58].valid := 1, [196].log_data[59].time := 3600.0, [196].log_data[59].valid := 1, [196].log_data[60].valid := 1, [196].log_data[61].valid := 1, [196].log_data[62].valid := 1, [196].log_data[63].valid := 1, [196].log_data[64].valid := 1, [196].log_data[65].valid := 1, [196].log_data[66].valid := 1, [196].log_data[67].valid := 1, [196].log_data[68].valid := 1, [196].log_data[69].valid := 1, [196].log_data[70].valid := 1, [196].log_data[71].valid := 1, [196].log_data[72].valid := 1, [196].log_data[73].valid := 1, [196].log_data[74].valid := 1, [196].log_data[75].valid := 1, [196].log_data[76].valid := 1, [196].log_data[77].valid := 1, [196].log_data[78].valid := 1, [196].log_data[79].valid := 1, [196].log_data[80].valid := 1, [196].log_data[81].valid := 1, [196].log_data[82].valid := 1,
        [196].log_data[83].valid := 1, [196].log_data[84].valid := 1, [196].log_data[85].valid := 1, [196].log_data[86].valid := 1, [196].log_data[87].valid := 1, [196].log_data[88].valid := 1, [196].log_data[89].valid := 1, [196].log_data[90].valid := 1, [196].log_data[91].valid := 1, [196].log_data[92].valid := 1, [196].log_data[93].valid := 1, [196].log_data[94].valid := 1, [196].log_data[95].valid := 1, [196].log_data[96].valid := 1, [196].log_data[97].valid := 1, [196].log_data[98].valid := 1, [196].log_data[99].valid := 1, [196].log_data[100].valid := 1, [196].log_data[101].valid := 1, [196].log_data[102].valid := 1, [196].log_data[103].valid := 1, [196].log_data[104].valid := 1, [196].log_data[105].valid := 1, [196].log_data[106].valid := 1, [196].log_data[107].valid := 1, [196].log_data[108].valid := 1, [196].log_data[109].valid := 1, [196].log_data[110].valid := 1, [196].log_data[111].valid := 1, [196].log_data[112].valid := 1, [196].log_data[113].valid := 1, [196].log_data[114].valid := 1, [196].log_data[115].valid := 1, [196].log_data[116].valid := 1, [196].log_data[117].valid := 1, [196].log_data[118].valid := 1, [196].log_data[119].valid := 1, [196].log_data[120].valid := 1, [196].log_data[121].valid := 1, [196].log_data[122].valid := 1, [196].log_data[123].valid := 1, [196].log_data[124].valid := 1, [196].time.Year := 2023, [196].time.Month := 1, [196].time.Day := 12, [196].time.Hour := 23, [196].time.Minute := 59, [196].time.Second := 59, [197].log_data[0].min := 1.0, [197].log_data[0].max := 1.0, [197].log_data[0].total := 3600.0, [197].log_data[0].time := 3600.0, [197].log_data[0].valid := 1, [197].log_data[1].max := 1.0, [197].log_data[1].total := 385.251, [197].log_data[1].time := 3600.0, [197].log_data[1].minminute := 6, [197].log_data[1].valid := 1, [197].log_data[2].max := 1.0, [197].log_data[2].total := 385.251,
        [197].log_data[2].time := 3600.0, [197].log_data[2].minminute := 6, [197].log_data[2].valid := 1, [197].log_data[3].time := 3600.0, [197].log_data[3].valid := 1, [197].log_data[4].time := 3600.0, [197].log_data[4].valid := 1, [197].log_data[5].max := 1.0, [197].log_data[5].total := 211.251, [197].log_data[5].time := 3600.0, [197].log_data[5].minminute := 1, [197].log_data[5].valid := 1, [197].log_data[6].time := 3600.0, [197].log_data[6].valid := 1, [197].log_data[7].time := 3600.0, [197].log_data[7].valid := 1, [197].log_data[8].min := 1.0, [197].log_data[8].max := 1.0, [197].log_data[8].total := 3600.0, [197].log_data[8].time := 3600.0, [197].log_data[8].valid := 1, [197].log_data[9].min := 1.0, [197].log_data[9].max := 1.0, [197].log_data[9].total := 3600.0, [197].log_data[9].time := 3600.0, [197].log_data[9].valid := 1, [197].log_data[10].min := 1.0, [197].log_data[10].max := 1.0, [197].log_data[10].total := 3600.0, [197].log_data[10].time := 3600.0, [197].log_data[10].valid := 1, [197].log_data[11].time := 3600.0, [197].log_data[11].valid := 1, [197].log_data[12].min := 1.0, [197].log_data[12].max := 1.0, [197].log_data[12].total := 3600.0, [197].log_data[12].time := 3600.0, [197].log_data[12].valid := 1, [197].log_data[13].min := 1.0, [197].log_data[13].max := 1.0, [197].log_data[13].total := 3600.0, [197].log_data[13].time := 3600.0, [197].log_data[13].valid := 1, [197].log_data[14].time := 3600.0, [197].log_data[14].valid := 1, [197].log_data[15].time := 3600.0, [197].log_data[15].valid := 1, [197].log_data[16].time := 3600.0, [197].log_data[16].valid := 1, [197].log_data[17].min := 1.0, [197].log_data[17].max := 1.0, [197].log_data[17].total := 3600.0, [197].log_data[17].time := 3600.0, [197].log_data[17].valid := 1, [197].log_data[18].time := 3600.0, [197].log_data[18].valid := 1, [197].log_data[19].time := 3600.0, [197].log_data[19].valid := 1, [197].log_data[20].time := 3600.0, [197].log_data[20].valid := 1,
        [197].log_data[21].min := 1.0, [197].log_data[21].max := 1.0, [197].log_data[21].total := 3600.0, [197].log_data[21].time := 3600.0, [197].log_data[21].valid := 1, [197].log_data[22].time := 3600.0, [197].log_data[22].valid := 1, [197].log_data[23].time := 3600.0, [197].log_data[23].valid := 1, [197].log_data[24].time := 3600.0, [197].log_data[24].valid := 1, [197].log_data[25].time := 3600.0, [197].log_data[25].valid := 1, [197].log_data[26].time := 3600.0, [197].log_data[26].valid := 1, [197].log_data[27].time := 3600.0, [197].log_data[27].valid := 1, [197].log_data[28].time := 3600.0, [197].log_data[28].valid := 1, [197].log_data[29].min := 1.0, [197].log_data[29].max := 1.0, [197].log_data[29].total := 3600.0, [197].log_data[29].time := 3600.0, [197].log_data[29].valid := 1, [197].log_data[30].min := 1.0, [197].log_data[30].max := 1.0, [197].log_data[30].total := 3600.0, [197].log_data[30].time := 3600.0, [197].log_data[30].valid := 1, [197].log_data[31].max := 1.0, [197].log_data[31].total := 1629.7471, [197].log_data[31].time := 3600.0, [197].log_data[31].valid := 1, [197].log_data[32].max := 1.0, [197].log_data[32].total := 1502.998, [197].log_data[32].time := 3600.0, [197].log_data[32].maxminute := 10, [197].log_data[32].valid := 1, [197].log_data[33].time := 3600.0, [197].log_data[33].valid := 1, [197].log_data[34].time := 3600.0, [197].log_data[34].valid := 1, [197].log_data[35].max := 1.0, [197].log_data[35].total := 1440.7471, [197].log_data[35].time := 3600.0, [197].log_data[35].minminute := 1, [197].log_data[35].valid := 1, [197].log_data[36].max := 1.0, [197].log_data[36].total := 1629.7471, [197].log_data[36].time := 3600.0, [197].log_data[36].maxminute := 3, [197].log_data[36].valid := 1, [197].log_data[37].max := 7.6109357, [197].log_data[37].total := 2425.2527, [197].log_data[37].time := 3600.0, [197].log_data[37].minminute := 5, [197].log_data[37].valid := 1, [197].log_data[38].time := 3600.0, [197].log_data[38].valid := 1, [197].log_data[39].min := 0.994824,
        [197].log_data[39].max := 1.0207345, [197].log_data[39].total := 3607.4915, [197].log_data[39].time := 3600.0, [197].log_data[39].minminute := 21, [197].log_data[39].maxminute := 3, [197].log_data[39].valid := 1, [197].log_data[40].min := 7.5673394, [197].log_data[40].max := 7.5805306, [197].log_data[40].total := 27267.986, [197].log_data[40].time := 3600.0, [197].log_data[40].minminute := 45, [197].log_data[40].maxminute := 26, [197].log_data[40].valid := 1, [197].log_data[41].min := 0.04727295, [197].log_data[41].max := 0.07514624, [197].log_data[41].total := 223.54108, [197].log_data[41].time := 3600.0, [197].log_data[41].minminute := 42, [197].log_data[41].maxminute := 29, [197].log_data[41].valid := 1, [197].log_data[42].min := 2.292585, [197].log_data[42].max := 2.2984736, [197].log_data[42].total := 8264.505, [197].log_data[42].time := 3600.0, [197].log_data[42].minminute := 5, [197].log_data[42].maxminute := 11, [197].log_data[42].valid := 1, [197].log_data[43].min := -0.26000214, [197].log_data[43].max := -0.23999786, [197].log_data[43].total := -935.9532, [197].log_data[43].time := 3600.0, [197].log_data[43].maxminute := 6, [197].log_data[43].valid := 1, [197].log_data[44].min := -0.30000305, [197].log_data[44].max := -0.27999878, [197].log_data[44].total := -1018.9041, [197].log_data[44].time := 3600.0, [197].log_data[44].minminute := 1, [197].log_data[44].valid := 1, [197].log_data[45].time := 3600.0, [197].log_data[45].valid := 1, [197].log_data[46].time := 3600.0, [197].log_data[46].valid := 1, [197].log_data[47].time := 3600.0, [197].log_data[47].valid := 1, [197].log_data[48].min := 6.578031, [197].log_data[48].max := 6.9649606, [197].log_data[48].total := 24238.002, [197].log_data[48].time := 3600.0, [197].log_data[48].minminute := 30, [197].log_data[48].maxminute := 6, [197].log_data[48].valid := 1, [197].log_data[49].min := 6.605368, [197].log_data[49].max := 9.306337, [197].log_data[49].total := 27925.799, [197].log_data[49].time := 3600.0, [197].log_data[49].minminute := 22, [197].log_data[49].valid := 1, [197].log_data[50].min := 2.0990808, [197].log_data[50].max := 2.1987183,
        [197].log_data[50].total := 7790.942, [197].log_data[50].time := 3600.0, [197].log_data[50].maxminute := 6, [197].log_data[50].valid := 1, [197].log_data[51].time := 3600.0, [197].log_data[51].valid := 1, [197].log_data[52].min := -3.1600037, [197].log_data[52].max := 0.11999512, [197].log_data[52].total := -7710.6523, [197].log_data[52].time := 3600.0, [197].log_data[52].minminute := 21, [197].log_data[52].valid := 1, [197].log_data[53].min := -2.5, [197].log_data[53].max := 0.22000122, [197].log_data[53].total := -7089.236, [197].log_data[53].time := 3600.0, [197].log_data[53].minminute := 50, [197].log_data[53].maxminute := 2, [197].log_data[53].valid := 1, [197].log_data[54].max := 0.572, [197].log_data[54].total := 1242.2124, [197].log_data[54].time := 3600.0, [197].log_data[54].maxminute := 21, [197].log_data[54].valid := 1, [197].log_data[55].max := 0.5345, [197].log_data[55].total := 1217.5532, [197].log_data[55].time := 3600.0, [197].log_data[55].minminute := 1, [197].log_data[55].maxminute := 34, [197].log_data[55].valid := 1, [197].log_data[56].min := 0.16024561, [197].log_data[56].max := 0.1607167, [197].log_data[56].total := 577.59, [197].log_data[56].time := 3600.0, [197].log_data[56].minminute := 21, [197].log_data[56].maxminute := 8, [197].log_data[56].valid := 1, [197].log_data[57].min := 0.32340303, [197].log_data[57].max := 0.32548368, [197].log_data[57].total := 1168.0526, [197].log_data[57].time := 3600.0, [197].log_data[57].minminute := 46, [197].log_data[57].maxminute := 8, [197].log_data[57].valid := 1, [197].log_data[58].time := 3600.0, [197].log_data[58].valid := 1, [197].log_data[59].time := 3600.0, [197].log_data[59].valid := 1, [197].log_data[60].valid := 1, [197].log_data[61].valid := 1, [197].log_data[62].valid := 1, [197].log_data[63].valid := 1, [197].log_data[64].valid := 1, [197].log_data[65].valid := 1, [197].log_data[66].valid := 1, [197].log_data[67].valid := 1, [197].log_data[68].valid := 1, [197].log_data[69].valid := 1, [197].log_data[70].valid := 1, [197].log_data[71].valid := 1,
        [197].log_data[72].valid := 1, [197].log_data[73].valid := 1, [197].log_data[74].valid := 1, [197].log_data[75].valid := 1, [197].log_data[76].valid := 1, [197].log_data[77].valid := 1, [197].log_data[78].valid := 1, [197].log_data[79].valid := 1, [197].log_data[80].valid := 1, [197].log_data[81].valid := 1, [197].log_data[82].valid := 1, [197].log_data[83].valid := 1, [197].log_data[84].valid := 1, [197].log_data[85].valid := 1, [197].log_data[86].valid := 1, [197].log_data[87].valid := 1, [197].log_data[88].valid := 1, [197].log_data[89].valid := 1, [197].log_data[90].valid := 1, [197].log_data[91].valid := 1, [197].log_data[92].valid := 1, [197].log_data[93].valid := 1, [197].log_data[94].valid := 1, [197].log_data[95].valid := 1, [197].log_data[96].valid := 1, [197].log_data[97].valid := 1, [197].log_data[98].valid := 1, [197].log_data[99].valid := 1, [197].log_data[100].valid := 1, [197].log_data[101].valid := 1, [197].log_data[102].valid := 1, [197].log_data[103].valid := 1, [197].log_data[104].valid := 1, [197].log_data[105].valid := 1, [197].log_data[106].valid := 1, [197].log_data[107].valid := 1, [197].log_data[108].valid := 1, [197].log_data[109].valid := 1, [197].log_data[110].valid := 1, [197].log_data[111].valid := 1, [197].log_data[112].valid := 1, [197].log_data[113].valid := 1, [197].log_data[114].valid := 1, [197].log_data[115].valid := 1, [197].log_data[116].valid := 1, [197].log_data[117].valid := 1, [197].log_data[118].valid := 1, [197].log_data[119].valid := 1, [197].log_data[120].valid := 1, [197].log_data[121].valid := 1, [197].log_data[122].valid := 1, [197].log_data[123].valid := 1, [197].log_data[124].valid := 1, [197].time.Year := 2023, [197].time.Month := 1, [197].time.Day := 13, [197].time.Minute := 59, [197].time.Second := 59, [198].log_data[0].min := 1.0, [198].log_data[0].max := 1.0,
        [198].log_data[0].total := 3599.5, [198].log_data[0].time := 3599.5, [198].log_data[0].valid := 1, [198].log_data[1].time := 3599.5, [198].log_data[1].valid := 1, [198].log_data[2].time := 3599.5, [198].log_data[2].valid := 1, [198].log_data[3].time := 3599.5, [198].log_data[3].valid := 1, [198].log_data[4].time := 3599.5, [198].log_data[4].valid := 1, [198].log_data[5].time := 3599.5, [198].log_data[5].valid := 1, [198].log_data[6].time := 3599.5, [198].log_data[6].valid := 1, [198].log_data[7].time := 3599.5, [198].log_data[7].valid := 1, [198].log_data[8].min := 1.0, [198].log_data[8].max := 1.0, [198].log_data[8].total := 3599.5, [198].log_data[8].time := 3599.5, [198].log_data[8].valid := 1, [198].log_data[9].min := 1.0, [198].log_data[9].max := 1.0, [198].log_data[9].total := 3599.5, [198].log_data[9].time := 3599.5, [198].log_data[9].valid := 1, [198].log_data[10].min := 1.0, [198].log_data[10].max := 1.0, [198].log_data[10].total := 3599.5, [198].log_data[10].time := 3599.5, [198].log_data[10].valid := 1, [198].log_data[11].time := 3599.5, [198].log_data[11].valid := 1, [198].log_data[12].min := 1.0, [198].log_data[12].max := 1.0, [198].log_data[12].total := 3599.5, [198].log_data[12].time := 3599.5, [198].log_data[12].valid := 1, [198].log_data[13].min := 1.0, [198].log_data[13].max := 1.0, [198].log_data[13].total := 3599.5, [198].log_data[13].time := 3599.5, [198].log_data[13].valid := 1, [198].log_data[14].time := 3599.5, [198].log_data[14].valid := 1, [198].log_data[15].time := 3599.5, [198].log_data[15].valid := 1, [198].log_data[16].time := 3599.5, [198].log_data[16].valid := 1, [198].log_data[17].min := 1.0, [198].log_data[17].max := 1.0, [198].log_data[17].total := 3599.5, [198].log_data[17].time := 3599.5, [198].log_data[17].valid := 1, [198].log_data[18].time := 3599.5, [198].log_data[18].valid := 1, [198].log_data[19].time := 3599.5, [198].log_data[19].valid := 1, [198].log_data[20].time := 3599.5,
        [198].log_data[20].valid := 1, [198].log_data[21].min := 1.0, [198].log_data[21].max := 1.0, [198].log_data[21].total := 3599.5, [198].log_data[21].time := 3599.5, [198].log_data[21].valid := 1, [198].log_data[22].time := 3599.5, [198].log_data[22].valid := 1, [198].log_data[23].time := 3599.5, [198].log_data[23].valid := 1, [198].log_data[24].time := 3599.5, [198].log_data[24].valid := 1, [198].log_data[25].time := 3599.5, [198].log_data[25].valid := 1, [198].log_data[26].time := 3599.5, [198].log_data[26].valid := 1, [198].log_data[27].time := 3599.5, [198].log_data[27].valid := 1, [198].log_data[28].time := 3599.5, [198].log_data[28].valid := 1, [198].log_data[29].min := 1.0, [198].log_data[29].max := 1.0, [198].log_data[29].total := 3599.5, [198].log_data[29].time := 3599.5, [198].log_data[29].valid := 1, [198].log_data[30].min := 1.0, [198].log_data[30].max := 1.0, [198].log_data[30].total := 3599.5, [198].log_data[30].time := 3599.5, [198].log_data[30].valid := 1, [198].log_data[31].max := 1.0, [198].log_data[31].total := 1629.7471, [198].log_data[31].time := 3599.5, [198].log_data[31].maxminute := 3, [198].log_data[31].valid := 1, [198].log_data[32].max := 1.0, [198].log_data[32].total := 1440.2471, [198].log_data[32].time := 3599.5, [198].log_data[32].minminute := 2, [198].log_data[32].valid := 1, [198].log_data[33].time := 3599.5, [198].log_data[33].valid := 1, [198].log_data[34].time := 3599.5, [198].log_data[34].valid := 1, [198].log_data[35].max := 1.0, [198].log_data[35].total := 1440.2471, [198].log_data[35].time := 3599.5, [198].log_data[35].minminute := 4, [198].log_data[35].valid := 1, [198].log_data[36].max := 1.0, [198].log_data[36].total := 1629.7471, [198].log_data[36].time := 3599.5, [198].log_data[36].maxminute := 6, [198].log_data[36].valid := 1, [198].log_data[37].time := 3599.5, [198].log_data[37].valid := 1, [198].log_data[38].time := 3599.5, [198].log_data[38].valid := 1, [198].log_data[39].min := 0.99529505, [198].log_data[39].max := 1.0060127,
        [198].log_data[39].total := 3603.488, [198].log_data[39].time := 3599.5, [198].log_data[39].minminute := 26, [198].log_data[39].maxminute := 3, [198].log_data[39].valid := 1, [198].log_data[40].min := 7.5673394, [198].log_data[40].max := 7.5794306, [198].log_data[40].total := 27267.385, [198].log_data[40].time := 3599.5, [198].log_data[40].minminute := 25, [198].log_data[40].maxminute := 9, [198].log_data[40].valid := 1, [198].log_data[41].min := 0.043346923, [198].log_data[41].max := 0.09143848, [198].log_data[41].total := 214.73145, [198].log_data[41].time := 3599.5, [198].log_data[41].minminute := 40, [198].log_data[41].maxminute := 8, [198].log_data[41].valid := 1, [198].log_data[42].min := 2.2921138, [198].log_data[42].max := 2.2990625, [198].log_data[42].total := 8263.724, [198].log_data[42].time := 3599.5, [198].log_data[42].minminute := 50, [198].log_data[42].maxminute := 27, [198].log_data[42].valid := 1, [198].log_data[43].min := -0.26000214, [198].log_data[43].max := -0.26000214, [198].log_data[43].total := -935.8432, [198].log_data[43].time := 3599.5, [198].log_data[43].valid := 1, [198].log_data[44].min := -0.30000305, [198].log_data[44].max := -0.27999878, [198].log_data[44].total := -1015.1146, [198].log_data[44].time := 3599.5, [198].log_data[44].valid := 1, [198].log_data[45].time := 3599.5, [198].log_data[45].valid := 1, [198].log_data[46].time := 3599.5, [198].log_data[46].valid := 1, [198].log_data[47].time := 3599.5, [198].log_data[47].valid := 1, [198].log_data[48].min := 6.7624273, [198].log_data[48].max := 6.7813888, [198].log_data[48].total := 24364.51, [198].log_data[48].time := 3599.5, [198].log_data[48].minminute := 59, [198].log_data[48].valid := 1, [198].log_data[49].min := 9.070984, [198].log_data[49].max := 9.3840685, [198].log_data[49].total := 33533.883, [198].log_data[49].time := 3599.5, [198].log_data[49].maxminute := 30, [198].log_data[49].valid := 1, [198].log_data[50].min := 2.045729, [198].log_data[50].max := 2.132882, [198].log_data[50].total := 7523.151, [198].log_data[50].time := 3599.5, [198].log_data[50].minminute := 58, [198].log_data[50].valid := 1,
        [198].log_data[51].time := 3599.5, [198].log_data[51].valid := 1, [198].log_data[52].min := -2.880005, [198].log_data[52].max := 0.11999512, [198].log_data[52].total := -7583.5815, [198].log_data[52].time := 3599.5, [198].log_data[52].minminute := 24, [198].log_data[52].maxminute := 2, [198].log_data[52].valid := 1, [198].log_data[53].min := -2.540001, [198].log_data[53].max := 0.19999695, [198].log_data[53].total := -7128.977, [198].log_data[53].time := 3599.5, [198].log_data[53].minminute := 18, [198].log_data[53].maxminute := 58, [198].log_data[53].valid := 1, [198].log_data[54].max := 0.5335, [198].log_data[54].total := 1216.9464, [198].log_data[54].time := 3599.5, [198].log_data[54].minminute := 2, [198].log_data[54].maxminute := 24, [198].log_data[54].valid := 1, [198].log_data[55].max := 0.5165, [198].log_data[55].total := 1216.9551, [198].log_data[55].time := 3599.5, [198].log_data[55].minminute := 4, [198].log_data[55].maxminute := 48, [198].log_data[55].valid := 1, [198].log_data[56].min := 0.16028486, [198].log_data[56].max := 0.1607167, [198].log_data[56].total := 577.62067, [198].log_data[56].time := 3599.5, [198].log_data[56].minminute := 8, [198].log_data[56].maxminute := 13, [198].log_data[56].valid := 1, [198].log_data[57].min := 0.32340303, [198].log_data[57].max := 0.32375634, [198].log_data[57].total := 1164.5858, [198].log_data[57].time := 3599.5, [198].log_data[57].minminute := 19, [198].log_data[57].maxminute := 4, [198].log_data[57].valid := 1, [198].log_data[58].time := 3599.5, [198].log_data[58].valid := 1, [198].log_data[59].time := 3599.5, [198].log_data[59].valid := 1, [198].log_data[60].valid := 1, [198].log_data[61].valid := 1, [198].log_data[62].valid := 1, [198].log_data[63].valid := 1, [198].log_data[64].valid := 1, [198].log_data[65].valid := 1, [198].log_data[66].valid := 1, [198].log_data[67].valid := 1, [198].log_data[68].valid := 1, [198].log_data[69].valid := 1, [198].log_data[70].valid := 1, [198].log_data[71].valid := 1, [198].log_data[72].valid := 1, [198].log_data[73].valid := 1,
        [198].log_data[74].valid := 1, [198].log_data[75].valid := 1, [198].log_data[76].valid := 1, [198].log_data[77].valid := 1, [198].log_data[78].valid := 1, [198].log_data[79].valid := 1, [198].log_data[80].valid := 1, [198].log_data[81].valid := 1, [198].log_data[82].valid := 1, [198].log_data[83].valid := 1, [198].log_data[84].valid := 1, [198].log_data[85].valid := 1, [198].log_data[86].valid := 1, [198].log_data[87].valid := 1, [198].log_data[88].valid := 1, [198].log_data[89].valid := 1, [198].log_data[90].valid := 1, [198].log_data[91].valid := 1, [198].log_data[92].valid := 1, [198].log_data[93].valid := 1, [198].log_data[94].valid := 1, [198].log_data[95].valid := 1, [198].log_data[96].valid := 1, [198].log_data[97].valid := 1, [198].log_data[98].valid := 1, [198].log_data[99].valid := 1, [198].log_data[100].valid := 1, [198].log_data[101].valid := 1, [198].log_data[102].valid := 1, [198].log_data[103].valid := 1, [198].log_data[104].valid := 1, [198].log_data[105].valid := 1, [198].log_data[106].valid := 1, [198].log_data[107].valid := 1, [198].log_data[108].valid := 1, [198].log_data[109].valid := 1, [198].log_data[110].valid := 1, [198].log_data[111].valid := 1, [198].log_data[112].valid := 1, [198].log_data[113].valid := 1, [198].log_data[114].valid := 1, [198].log_data[115].valid := 1, [198].log_data[116].valid := 1, [198].log_data[117].valid := 1, [198].log_data[118].valid := 1, [198].log_data[119].valid := 1, [198].log_data[120].valid := 1, [198].log_data[121].valid := 1, [198].log_data[122].valid := 1, [198].log_data[123].valid := 1, [198].log_data[124].valid := 1, [198].time.Year := 2023, [198].time.Month := 1, [198].time.Day := 13, [198].time.Hour := 1, [198].time.Minute := 59, [198].time.Second := 59, [199].log_data[0].min := 1.0, [199].log_data[0].max := 1.0, [199].log_data[0].total := 3600.0,
        [199].log_data[0].time := 3600.0, [199].log_data[0].valid := 1, [199].log_data[1].max := 1.0, [199].log_data[1].total := 563.0, [199].log_data[1].time := 3600.0, [199].log_data[1].maxminute := 9, [199].log_data[1].valid := 1, [199].log_data[2].max := 1.0, [199].log_data[2].total := 559.5, [199].log_data[2].time := 3600.0, [199].log_data[2].maxminute := 9, [199].log_data[2].valid := 1, [199].log_data[3].time := 3600.0, [199].log_data[3].valid := 1, [199].log_data[4].time := 3600.0, [199].log_data[4].valid := 1, [199].log_data[5].max := 1.0, [199].log_data[5].total := 227.5, [199].log_data[5].time := 3600.0, [199].log_data[5].maxminute := 11, [199].log_data[5].valid := 1, [199].log_data[6].time := 3600.0, [199].log_data[6].valid := 1, [199].log_data[7].time := 3600.0, [199].log_data[7].valid := 1, [199].log_data[8].min := 1.0, [199].log_data[8].max := 1.0, [199].log_data[8].total := 3600.0, [199].log_data[8].time := 3600.0, [199].log_data[8].valid := 1, [199].log_data[9].min := 1.0, [199].log_data[9].max := 1.0, [199].log_data[9].total := 3600.0, [199].log_data[9].time := 3600.0, [199].log_data[9].valid := 1, [199].log_data[10].min := 1.0, [199].log_data[10].max := 1.0, [199].log_data[10].total := 3600.0, [199].log_data[10].time := 3600.0, [199].log_data[10].valid := 1, [199].log_data[11].time := 3600.0, [199].log_data[11].valid := 1, [199].log_data[12].min := 1.0, [199].log_data[12].max := 1.0, [199].log_data[12].total := 3600.0, [199].log_data[12].time := 3600.0, [199].log_data[12].valid := 1, [199].log_data[13].min := 1.0, [199].log_data[13].max := 1.0, [199].log_data[13].total := 3600.0, [199].log_data[13].time := 3600.0, [199].log_data[13].valid := 1, [199].log_data[14].time := 3600.0, [199].log_data[14].valid := 1, [199].log_data[15].time := 3600.0, [199].log_data[15].valid := 1, [199].log_data[16].time := 3600.0, [199].log_data[16].valid := 1, [199].log_data[17].min := 1.0, [199].log_data[17].max := 1.0,
        [199].log_data[17].total := 3600.0, [199].log_data[17].time := 3600.0, [199].log_data[17].valid := 1, [199].log_data[18].time := 3600.0, [199].log_data[18].valid := 1, [199].log_data[19].time := 3600.0, [199].log_data[19].valid := 1, [199].log_data[20].time := 3600.0, [199].log_data[20].valid := 1, [199].log_data[21].min := 1.0, [199].log_data[21].max := 1.0, [199].log_data[21].total := 3600.0, [199].log_data[21].time := 3600.0, [199].log_data[21].valid := 1, [199].log_data[22].time := 3600.0, [199].log_data[22].valid := 1, [199].log_data[23].time := 3600.0, [199].log_data[23].valid := 1, [199].log_data[24].time := 3600.0, [199].log_data[24].valid := 1, [199].log_data[25].time := 3600.0, [199].log_data[25].valid := 1, [199].log_data[26].time := 3600.0, [199].log_data[26].valid := 1, [199].log_data[27].time := 3600.0, [199].log_data[27].valid := 1, [199].log_data[28].time := 3600.0, [199].log_data[28].valid := 1, [199].log_data[29].min := 1.0, [199].log_data[29].max := 1.0, [199].log_data[29].total := 3600.0, [199].log_data[29].time := 3600.0, [199].log_data[29].valid := 1, [199].log_data[30].min := 1.0, [199].log_data[30].max := 1.0, [199].log_data[30].total := 3600.0, [199].log_data[30].time := 3600.0, [199].log_data[30].valid := 1, [199].log_data[31].max := 1.0, [199].log_data[31].total := 1629.7471, [199].log_data[31].time := 3600.0, [199].log_data[31].maxminute := 6, [199].log_data[31].valid := 1, [199].log_data[32].max := 1.0, [199].log_data[32].total := 1440.998, [199].log_data[32].time := 3600.0, [199].log_data[32].minminute := 5, [199].log_data[32].valid := 1, [199].log_data[33].time := 3600.0, [199].log_data[33].valid := 1, [199].log_data[34].time := 3600.0, [199].log_data[34].valid := 1, [199].log_data[35].max := 1.0, [199].log_data[35].total := 1568.498, [199].log_data[35].time := 3600.0, [199].log_data[35].minminute := 8, [199].log_data[35].valid := 1, [199].log_data[36].max := 1.0, [199].log_data[36].total := 1584.998, [199].log_data[36].time := 3600.0,
        [199].log_data[36].maxminute := 9, [199].log_data[36].valid := 1, [199].log_data[37].max := 7.1610355, [199].log_data[37].total := 3433.5674, [199].log_data[37].time := 3600.0, [199].log_data[37].maxminute := 12, [199].log_data[37].valid := 1, [199].log_data[38].time := 3600.0, [199].log_data[38].valid := 1, [199].log_data[39].min := 0.9957663, [199].log_data[39].max := 1.0213233, [199].log_data[39].total := 3609.9546, [199].log_data[39].time := 3600.0, [199].log_data[39].minminute := 27, [199].log_data[39].maxminute := 15, [199].log_data[39].valid := 1, [199].log_data[40].min := 7.555797, [199].log_data[40].max := 7.586026, [199].log_data[40].total := 27266.898, [199].log_data[40].time := 3600.0, [199].log_data[40].minminute := 1, [199].log_data[40].maxminute := 6, [199].log_data[40].valid := 1, [199].log_data[41].min := 0.05335791, [199].log_data[41].max := 0.08319409, [199].log_data[41].total := 233.2469, [199].log_data[41].time := 3600.0, [199].log_data[41].minminute := 38, [199].log_data[41].maxminute := 52, [199].log_data[41].valid := 1, [199].log_data[42].min := 2.292467, [199].log_data[42].max := 2.3001225, [199].log_data[42].total := 8264.767, [199].log_data[42].time := 3600.0, [199].log_data[42].minminute := 3, [199].log_data[42].maxminute := 54, [199].log_data[42].valid := 1, [199].log_data[43].min := -0.26000214, [199].log_data[43].max := -0.26000214, [199].log_data[43].total := -935.9732, [199].log_data[43].time := 3600.0, [199].log_data[43].valid := 1, [199].log_data[44].min := -0.30000305, [199].log_data[44].max := -0.27999878, [199].log_data[44].total := -1047.1312, [199].log_data[44].time := 3600.0, [199].log_data[44].valid := 1, [199].log_data[45].time := 3600.0, [199].log_data[45].valid := 1, [199].log_data[46].time := 3600.0, [199].log_data[46].valid := 1, [199].log_data[47].time := 3600.0, [199].log_data[47].valid := 1, [199].log_data[48].min := 6.581329, [199].log_data[48].max := 6.969357, [199].log_data[48].total := 24236.244, [199].log_data[48].time := 3600.0, [199].log_data[48].minminute := 41, [199].log_data[48].maxminute := 13, [199].log_data[48].valid := 1,
        [199].log_data[49].min := 6.7315836, [199].log_data[49].max := 9.384853, [199].log_data[49].total := 28831.795, [199].log_data[49].time := 3600.0, [199].log_data[49].minminute := 38, [199].log_data[49].maxminute := 6, [199].log_data[49].valid := 1, [199].log_data[50].min := 2.0307715, [199].log_data[50].max := 2.1314688, [199].log_data[50].total := 7524.4194, [199].log_data[50].time := 3600.0, [199].log_data[50].minminute := 10, [199].log_data[50].maxminute := 19, [199].log_data[50].valid := 1, [199].log_data[51].time := 3600.0, [199].log_data[51].valid := 1, [199].log_data[52].min := -2.880005, [199].log_data[52].max := 0.11999512, [199].log_data[52].total := -7624.7803, [199].log_data[52].time := 3600.0, [199].log_data[52].minminute := 27, [199].log_data[52].maxminute := 5, [199].log_data[52].valid := 1, [199].log_data[53].min := -2.5200043, [199].log_data[53].max := 0.19999695, [199].log_data[53].total := -7394.368, [199].log_data[53].time := 3600.0, [199].log_data[53].minminute := 10, [199].log_data[53].maxminute := 40, [199].log_data[53].valid := 1, [199].log_data[54].max := 0.5295, [199].log_data[54].total := 1217.4423, [199].log_data[54].time := 3600.0, [199].log_data[54].minminute := 5, [199].log_data[54].maxminute := 27, [199].log_data[54].valid := 1, [199].log_data[55].max := 0.538, [199].log_data[55].total := 1252.144, [199].log_data[55].time := 3600.0, [199].log_data[55].minminute := 8, [199].log_data[55].maxminute := 30, [199].log_data[55].valid := 1, [199].log_data[56].min := 0.16028486, [199].log_data[56].max := 0.1607167, [199].log_data[56].total := 577.6272, [199].log_data[56].time := 3600.0, [199].log_data[56].minminute := 37, [199].log_data[56].valid := 1, [199].log_data[57].min := 0.32202896, [199].log_data[57].max := 0.3237171, [199].log_data[57].total := 1163.263, [199].log_data[57].time := 3600.0, [199].log_data[57].minminute := 51, [199].log_data[57].valid := 1, [199].log_data[58].time := 3600.0, [199].log_data[58].valid := 1, [199].log_data[59].time := 3600.0, [199].log_data[59].valid := 1, [199].log_data[60].valid := 1, [199].log_data[61].valid := 1,
        [199].log_data[62].valid := 1, [199].log_data[63].valid := 1, [199].log_data[64].valid := 1, [199].log_data[65].valid := 1, [199].log_data[66].valid := 1, [199].log_data[67].valid := 1, [199].log_data[68].valid := 1, [199].log_data[69].valid := 1, [199].log_data[70].valid := 1, [199].log_data[71].valid := 1, [199].log_data[72].valid := 1, [199].log_data[73].valid := 1, [199].log_data[74].valid := 1, [199].log_data[75].valid := 1, [199].log_data[76].valid := 1, [199].log_data[77].valid := 1, [199].log_data[78].valid := 1, [199].log_data[79].valid := 1, [199].log_data[80].valid := 1, [199].log_data[81].valid := 1, [199].log_data[82].valid := 1, [199].log_data[83].valid := 1, [199].log_data[84].valid := 1, [199].log_data[85].valid := 1, [199].log_data[86].valid := 1, [199].log_data[87].valid := 1, [199].log_data[88].valid := 1, [199].log_data[89].valid := 1, [199].log_data[90].valid := 1, [199].log_data[91].valid := 1, [199].log_data[92].valid := 1, [199].log_data[93].valid := 1, [199].log_data[94].valid := 1, [199].log_data[95].valid := 1, [199].log_data[96].valid := 1, [199].log_data[97].valid := 1, [199].log_data[98].valid := 1, [199].log_data[99].valid := 1, [199].log_data[100].valid := 1, [199].log_data[101].valid := 1, [199].log_data[102].valid := 1, [199].log_data[103].valid := 1, [199].log_data[104].valid := 1, [199].log_data[105].valid := 1, [199].log_data[106].valid := 1, [199].log_data[107].valid := 1, [199].log_data[108].valid := 1, [199].log_data[109].valid := 1, [199].log_data[110].valid := 1, [199].log_data[111].valid := 1, [199].log_data[112].valid := 1, [199].log_data[113].valid := 1, [199].log_data[114].valid := 1, [199].log_data[115].valid := 1, [199].log_data[116].valid := 1, [199].log_data[117].valid := 1, [199].log_data[118].valid := 1, [199].log_data[119].valid := 1, [199].log_data[120].valid := 1, [199].log_data[121].valid := 1,
        [199].log_data[122].valid := 1, [199].log_data[123].valid := 1, [199].log_data[124].valid := 1, [199].time.Year := 2023, [199].time.Month := 1, [199].time.Day := 13, [199].time.Hour := 2, [199].time.Minute := 59, [199].time.Second := 59);
   report_pwrup_done : BOOL := 1;
   report_row_daily : DINT := 156;
   report_row_qty : DINT := 200;
   report_tag_qty : DINT := 125;
   SCR201 : MOTOR := (fail_dlay := 60, start_dlay := 3000, auto := 1, remote := 1, permit := 1, run_sts := 1, run_out := 1, runtime := 1929.584, runtime_f := 0.58400255, runtime_i := 1929, fail_tonr.TimerEnable := 1, fail_tonr.PRE := 60000, fail_tonr.Reset := 1, start_os.InputBit := 1, manual_mode_timer.Reset := 1);   // Inlet screen 1 brush motor
   SCR202 : MOTOR := (fail_dlay := 60, start_dlay := 3000, auto := 1, remote := 1, permit := 1, run_sts := 1, run_out := 1, runtime := 1912.9653, runtime_f := 0.9653193, runtime_i := 1912, fail_tonr.TimerEnable := 1, fail_tonr.PRE := 60000, fail_tonr.Reset := 1, start_os.InputBit := 1, manual_mode_timer.Reset := 1);   // Inlet screen 2 brush motor
   VIT701 : PRANALOG := (MinEU := -100.0, MaxEU := 100.0, lolim := -20.0, lololim := -20.0, raw := 4990.0, calc := -0.19999695, value := -0.19999695, valid := 1, log := 1);   // Membrane tank 1 vacuum pressure
   VIT702 : PRANALOG := (MinEU := -100.0, MaxEU := 100.0, lolim := -8.0, lololim := -10.0, raw := 4989.0, calc := -0.22000122, value := -0.22000122, valid := 1, log := 1);   // Membrane tank 2 vacuum pressure
   VIT703 : PRANALOG := (MinEU := -100.0, MaxEU := 100.0, lolim := -20.0, lololim := -20.0, raw := 4928.0, calc := -1.4400024, value := -1.4400024, valid := 1, log := 1);   // Membrane tank 3 vacuum pressure
   VIT704 : PRANALOG := (MinEU := -100.0, MaxEU := 100.0, lolim := -20.0, lololim := -20.0, raw := 4931.0, calc := -1.3800049, value := -1.3800049, valid := 1, log := 1);   // Membrane tank 4 vacuum pressure
   WALLCLOCK : DateTime := (Year := 2023, Month := 1, Day := 19, Hour := 15, Minute := 26, Second := 5, Microsecond := 9024, DayOfWeek := 4);   // Global date / time
   WALLCLOCK_lock : BOOL;
END_VAR
